{attribute addProperty BoxType "EK1100-0000-0018"}
{attribute addProperty Id "Beckhoff_EJx9xxEK1122Beckhoff_EJx9xxEK1122_05D2B413162A_0001_EJ1914_0000_0017EJ1914_5EB96E2D21026.25A_0002_EJ1914_0000_0018EJ1914_5EB96E2D21026.25A_0003_EJ1918_0000_0017EJ1918_151E5A8221827.25A_0004_EJ1918_0000_0018EJ1918_151E5A8221827.25A_0005_EJ1957_0000_0017EJ1957_6B6926D126032.5A_0006_EJ1957_0000_0018EJ1957_6B6926D126032.5A_0007_EJ2914_0000_0017EJ2914_46D107EB24430.5A_0008_EJ2914_0000_0018EJ2914_46D107EB24430.5A_0009_EJ2918_0000_0017EJ2918_AA36864B28435.5A_0010_EJ2918_0000_0018EJ2918_AA36864B28435.5A_0011_EJ6910_0000_0018EJ6910_4EA245C69812.25A_0012_EJ6910_0000_0020EJ6910_4EA245C69812.25"}
{attribute addProperty CRC "2836563209"}
{attribute addProperty SizeInBites "2644"}
{attribute addProperty SizeInBytes "330.5"}
TYPE Beckhoff_EJx9xx_A9128509 EXTENDS EK1100_179A0949 :
STRUCT
	{attribute addProperty Name "Beckhoff_EJx9xxEK1122"}
	Beckhoff_EJx9xxEK1122 : Beckhoff_EJx9xxEK1122_05D2B413;
	{attribute addProperty Name "A_0001_EJ1914_0000_0017"}
	A_0001_EJ1914_0000_0017 : EJ1914_5EB96E2D;
	{attribute addProperty Name "A_0002_EJ1914_0000_0018"}
	A_0002_EJ1914_0000_0018 : EJ1914_5EB96E2D;
	{attribute addProperty Name "A_0003_EJ1918_0000_0017"}
	A_0003_EJ1918_0000_0017 : EJ1918_151E5A82;
	{attribute addProperty Name "A_0004_EJ1918_0000_0018"}
	A_0004_EJ1918_0000_0018 : EJ1918_151E5A82;
	{attribute addProperty Name "A_0005_EJ1957_0000_0017"}
	A_0005_EJ1957_0000_0017 : EJ1957_6B6926D1;
	{attribute addProperty Name "A_0006_EJ1957_0000_0018"}
	A_0006_EJ1957_0000_0018 : EJ1957_6B6926D1;
	{attribute addProperty Name "A_0007_EJ2914_0000_0017"}
	A_0007_EJ2914_0000_0017 : EJ2914_46D107EB;
	{attribute addProperty Name "A_0008_EJ2914_0000_0018"}
	A_0008_EJ2914_0000_0018 : EJ2914_46D107EB;
	{attribute addProperty Name "A_0009_EJ2918_0000_0017"}
	A_0009_EJ2918_0000_0017 : EJ2918_AA36864B;
	{attribute addProperty Name "A_0010_EJ2918_0000_0018"}
	A_0010_EJ2918_0000_0018 : EJ2918_AA36864B;
	{attribute addProperty Name "A_0011_EJ6910_0000_0018"}
	A_0011_EJ6910_0000_0018 : EJ6910_4EA245C6;
	{attribute addProperty Name "A_0012_EJ6910_0000_0020"}
	A_0012_EJ6910_0000_0020 : EJ6910_4EA245C6;
END_STRUCT
END_TYPE

(* stored: Version 1.2.0.0, ProductVersion 3.1.4024.9
   DUT Beckhoff_EJx9xx_A9128509: Id {407a933f-4d1b-48e2-bfa3-114e4141fd93} *)
